{attribute addProperty BoxType "KL2535-0001"}
{attribute addProperty Id "Channel_100Channel_200"}
{attribute addProperty CRC "2989660623"}
{attribute addProperty SizeInBites "0"}
{attribute addProperty SizeInBytes "0"}
TYPE KL_B23299CF :
STRUCT
	{attribute addProperty Name "Channel_1"}
	Channel_1 : ;
	{attribute addProperty Name "Channel_2"}
	Channel_2 : ;
END_STRUCT
END_TYPE

(* stored: Version 1.2.0.0, ProductVersion 3.1.4024.9
   DUT KL_B23299CF: Id {175ae608-20c2-4210-9fa2-107476eb4119} *)
